	DATA_BLOCK DB376
	TITLE =DBG276M  HEATING KILN 1
	//COPYRIGHT:    (C) 2009  BUHLER AG, CH-9240 UZWIL, SWITZERLAND
	//
	//PRODUCT:      WinCoS_BIW01_09
	//
	//TITLE:        HEATING KILN 1
	//                Machine group DB
	//                Maschinengruppen-DB
	//
	//-------------------------------------------------------------------------
	//
	//IDENT:        AUTHOR:             DEPT:             DATE:
	//
	//P01_DB376.1.0 K.Renz              CSB41             13.Jan.2010
	//              1st Release
	//
	//-------------------------------------------------------------------------
	//
	//PURPOSE:
	//
	//MANUAL :
	//
	//RESTRICTIONS:
	//
	//-------------------------------------------------------------------------
	AUTHOR  : KR
	FAMILY  : USW
	NAME    : DBG276M
	VERSION : 00.00

	FB376
	BEGIN
	      #Gr.Par.ParObjectNo 	:=27600;
	      #Gr.Par.ParIdling      	:=2;
	      #Gr.Par.ParMgr	        :=True;
	      #Gr.Par.ParWgr	        :=False;
	      #Gr.Par.ParGgr	        :=False;
	      #Gr.Par.ParEmptyingTime 	:=0;
	      #Gr.Par.ParHornCode       :=10;
	//Parameter =A-3191-BPS21 : HEAT EXCHANGE PRESSURE < 15mbar
	      #A_3191_BPS21.Par.ParObjectNo                             :=27601;
	      #A_3191_BPS21.Par.ParMsgType                              :=7154;
	      #A_3191_BPS21.Par.ParHornCode                             :=10;
	      #A_3191_BPS21.Par.ParDelayChange                          :=20;
	      #A_3191_BPS21.Par.ParDelayTrue                            :=10;
	      #A_3191_BPS21.Par.ParDelayFalse                           :=0;
	      #A_3191_BPS21.Par.ParTimeoutTrue                          :=0;
	      #A_3191_BPS21.Par.ParTimeoutFalse                         :=0;
	      #A_3191_BPS21.Par.ParLogOff                               :=False;
	      #A_3191_BPS21.Par.Par2WorkingCond                         :=False;
	      #A_3191_BPS21.Par.ParFaultRetry                           :=False;
	      #A_3191_BPS21.Par.ParBinLevel                             :=False;
	//
	//
	//Parameter =A-3161-KCL12 : BURNER 2 ALARM SUMMARY
	      #A_3161_KCL12.Par.ParObjectNo                             :=27602;
	      #A_3161_KCL12.Par.ParMsgType                              :=7154;
	      #A_3161_KCL12.Par.ParHornCode                             :=10;
	      #A_3161_KCL12.Par.ParDelayChange                          :=20;
	      #A_3161_KCL12.Par.ParDelayTrue                            :=10;
	      #A_3161_KCL12.Par.ParDelayFalse                           :=0;
	      #A_3161_KCL12.Par.ParTimeoutTrue                          :=0;
	      #A_3161_KCL12.Par.ParTimeoutFalse                         :=0;
	      #A_3161_KCL12.Par.ParLogOff                               :=False;
	      #A_3161_KCL12.Par.Par2WorkingCond                         :=False;
	      #A_3161_KCL12.Par.ParFaultRetry                           :=False;
	      #A_3161_KCL12.Par.ParBinLevel                             :=False;
	//
	//
	//Parameter =A-3161-KCL12_EXT_ON : BURNER 2 EXTERAL ON
	      #A_3161_KCL12_EXT_ON.Par.ParObjectNo                             :=27603;
	      #A_3161_KCL12_EXT_ON.Par.ParMsgType                              :=7002;
	      #A_3161_KCL12_EXT_ON.Par.ParHornCode                             :=0;
	      #A_3161_KCL12_EXT_ON.Par.ParOnTime                               :=10;
	      #A_3161_KCL12_EXT_ON.Par.ParOffTime                              :=0;
	      #A_3161_KCL12_EXT_ON.Par.ParIdlingTime                           :=0;
	      #A_3161_KCL12_EXT_ON.Par.ParDelayTime                            :=0;
	      #A_3161_KCL12_EXT_ON.Par.ParLogOff                               :=False;
	      #A_3161_KCL12_EXT_ON.Par.ParManual                               :=True;
	      #A_3161_KCL12_EXT_ON.Par.ParContinuous                           :=True;
	      #A_3161_KCL12_EXT_ON.Par.ParPulse                                :=False;
	      #A_3161_KCL12_EXT_ON.Par.ParPulsing                              :=False;
	      #A_3161_KCL12_EXT_ON.Par.ParFilter                               :=False;
	//
	//
	//Parameter =A-3161-KCL12_ON : BURNER 2 ON
	      #A_3161_KCL12_ON.Par.ParObjectNo                             :=27604;
	      #A_3161_KCL12_ON.Par.ParMsgType                              :=7154;
	      #A_3161_KCL12_ON.Par.ParHornCode                             :=0;
	      #A_3161_KCL12_ON.Par.ParDelayChange                          :=20;
	      #A_3161_KCL12_ON.Par.ParDelayTrue                            :=10;
	      #A_3161_KCL12_ON.Par.ParDelayFalse                           :=0;
	      #A_3161_KCL12_ON.Par.ParTimeoutTrue                          :=0;
	      #A_3161_KCL12_ON.Par.ParTimeoutFalse                         :=0;
	      #A_3161_KCL12_ON.Par.ParLogOff                               :=False;
	      #A_3161_KCL12_ON.Par.Par2WorkingCond                         :=False;
	      #A_3161_KCL12_ON.Par.ParFaultRetry                           :=False;
	      #A_3161_KCL12_ON.Par.ParBinLevel                             :=False;
	//
	//
	//Parameter =A-3161-KCL12_RUN : BURNER 2 MAIN FAN RUNNING
	      #A_3161_KCL12_RUN.Par.ParObjectNo                             :=27609;
	      #A_3161_KCL12_RUN.Par.ParMsgType                              :=7002;
	      #A_3161_KCL12_RUN.Par.ParHornCode                             :=0;
	      #A_3161_KCL12_RUN.Par.ParOnTime                               :=10;
	      #A_3161_KCL12_RUN.Par.ParOffTime                              :=0;
	      #A_3161_KCL12_RUN.Par.ParIdlingTime                           :=0;
	      #A_3161_KCL12_RUN.Par.ParDelayTime                            :=0;
	      #A_3161_KCL12_RUN.Par.ParLogOff                               :=False;
	      #A_3161_KCL12_RUN.Par.ParManual                               :=True;
	      #A_3161_KCL12_RUN.Par.ParContinuous                           :=True;
	      #A_3161_KCL12_RUN.Par.ParPulse                                :=False;
	      #A_3161_KCL12_RUN.Par.ParPulsing                              :=False;
	      #A_3161_KCL12_RUN.Par.ParFilter                               :=False;
	//
	//
	//Parameter =A-3161-KCL12_AI : BURNER 2 INPUT SIGNAL ANALOG
	      #A_3161_KCL12_AI.Par.ParObjectNo                             :=27605;
	      #A_3161_KCL12_AI.Par.ParHornCode                             :=10;
	      #A_3161_KCL12_AI.Par.ParMsgType                              :=7252;
	      #A_3161_KCL12_AI.Par.ParUnitsByZeroDigit                     :=L#0;
	      #A_3161_KCL12_AI.Par.ParUnitsByMaxDigit                      :=L#16384;
	      #A_3161_KCL12_AI.Par.ParUnitsBy100Pc                         :=L#10000;
	      #A_3161_KCL12_AI.Par.ParDelayTimeDown                        :=10;
	      #A_3161_KCL12_AI.Par.ParDelayTimeUp                          :=10;
	      #A_3161_KCL12_AI.Par.ParDelayTime                            :=30;
	      #A_3161_KCL12_AI.Par.ParLimitLL                              :=L#-1;
	      #A_3161_KCL12_AI.Par.ParLimitL                               :=L#0;
	      #A_3161_KCL12_AI.Par.ParLimitH                               :=L#7000;
	      #A_3161_KCL12_AI.Par.ParLimitHH                              :=L#8000;
	      #A_3161_KCL12_AI.Par.ParMonTimeLL                            :=0;
	      #A_3161_KCL12_AI.Par.ParMonTimeL                             :=0;
	      #A_3161_KCL12_AI.Par.ParMonTimeMid                           :=0;
	      #A_3161_KCL12_AI.Par.ParMonTimeH                             :=0;
	      #A_3161_KCL12_AI.Par.ParMonTimeHH                            :=0;
	      #A_3161_KCL12_AI.Par.ParLogOff                               :=False;
	      #A_3161_KCL12_AI.Par.ParValueByUser                          :=False;
	      #A_3161_KCL12_AI.Par.ParLimitsPc                             :=True;
	      #A_3161_KCL12_AI.Par.ParWago                                 :=False;
	      #A_3161_KCL12_AI.Par.ParNoHornByWarning                      :=False;
	      #A_3161_KCL12_AI.Par.ParWarningLL                            :=False;
	      #A_3161_KCL12_AI.Par.ParWarningL                             :=False;
	      #A_3161_KCL12_AI.Par.ParWarningMid                           :=False;
	      #A_3161_KCL12_AI.Par.ParWarningH                             :=False;
	      #A_3161_KCL12_AI.Par.ParWarningHH                            :=False;
	      #A_3161_KCL12_AI.Par.ParPreAlarmLL                           :=False;
	      #A_3161_KCL12_AI.Par.ParPreAlarmL                            :=False;
	      #A_3161_KCL12_AI.Par.ParPreAlarmMid                          :=False;
	      #A_3161_KCL12_AI.Par.ParPreAlarmH                            :=False;
	      #A_3161_KCL12_AI.Par.ParPreAlarmHH                           :=False;
	//
	//
	//Parameter =A-3161-KCL12_AO : BURNER 2 OUTPUT SIGNAL ANALOG
	      #A_3161_KCL12_AO.Par.ParObjectNo                             :=27606;
	      #A_3161_KCL12_AO.Par.ParMsgType                              :=7241;
	      #A_3161_KCL12_AO.Par.ParHornCode                             :=10;
	      #A_3161_KCL12_AO.Par.ParUnitsByZeroDigit                     :=L#0;
	      #A_3161_KCL12_AO.Par.ParUnitsByMaxDigit                      :=L#27648;
	      #A_3161_KCL12_AO.Par.ParUnitsBy100Pc                         :=L#10000;
	      #A_3161_KCL12_AO.Par.ParLimitMin                             :=L#0;
	      #A_3161_KCL12_AO.Par.ParLimitMax                             :=L#27648;
	      #A_3161_KCL12_AO.Par.ParDelayTime                            :=30;
	      #A_3161_KCL12_AO.Par.ParLogOff                               :=False;
	      #A_3161_KCL12_AO.Par.ParValuePc                              :=True;
	      #A_3161_KCL12_AO.Par.ParLimitsPc                             :=True;
	      #A_3161_KCL12_AO.Par.ParWago                                 :=False;
	      #A_3161_KCL12_AO.Par.ParFU                                   :=False;
	//
	//
	//Parameter =A-3161-KCL12_REG_ON : BURNER 2 REGULATOR ON
	      #A_3161_KCL12_REG_ON.Par.ParObjectNo                             :=27607;
	      #A_3161_KCL12_REG_ON.Par.ParMsgType                              :=7154;
	      #A_3161_KCL12_REG_ON.Par.ParHornCode                             :=10;
	      #A_3161_KCL12_REG_ON.Par.ParDelayChange                          :=20;
	      #A_3161_KCL12_REG_ON.Par.ParDelayTrue                            :=10;
	      #A_3161_KCL12_REG_ON.Par.ParDelayFalse                           :=0;
	      #A_3161_KCL12_REG_ON.Par.ParTimeoutTrue                          :=0;
	      #A_3161_KCL12_REG_ON.Par.ParTimeoutFalse                         :=0;
	      #A_3161_KCL12_REG_ON.Par.ParLogOff                               :=False;
	      #A_3161_KCL12_REG_ON.Par.Par2WorkingCond                         :=False;
	      #A_3161_KCL12_REG_ON.Par.ParFaultRetry                           :=False;
	      #A_3161_KCL12_REG_ON.Par.ParBinLevel                             :=False;
	//
	//
	//Parameter =A-3161-KCL12_REM_OP : BURNER 2 REMOTE OPERATION
	      #A_3161_KCL12_REM_OP.Par.ParObjectNo                             :=27608;
	      #A_3161_KCL12_REM_OP.Par.ParMsgType                              :=7154;
	      #A_3161_KCL12_REM_OP.Par.ParHornCode                             :=10;
	      #A_3161_KCL12_REM_OP.Par.ParDelayChange                          :=20;
	      #A_3161_KCL12_REM_OP.Par.ParDelayTrue                            :=10;
	      #A_3161_KCL12_REM_OP.Par.ParDelayFalse                           :=0;
	      #A_3161_KCL12_REM_OP.Par.ParTimeoutTrue                          :=0;
	      #A_3161_KCL12_REM_OP.Par.ParTimeoutFalse                         :=0;
	      #A_3161_KCL12_REM_OP.Par.ParLogOff                               :=False;
	      #A_3161_KCL12_REM_OP.Par.Par2WorkingCond                         :=False;
	      #A_3161_KCL12_REM_OP.Par.ParFaultRetry                           :=False;
	      #A_3161_KCL12_REM_OP.Par.ParBinLevel                             :=False;
	//
	//
	END_DATA_BLOCK
